TEXTLIST TL_LOG_LEVEL
  0 = 'TRACE'
  1 = 'DEBUG'
  2 = 'INFO'
  3 = 'WARN'
  4 = 'ERROR'
  5 = 'OFF'
   = ''
END_TEXTLIST

(* stored: Version 1.1.0.1, ProductVersion 3.1.4026.18
   TextList TL_LOG_LEVEL: Id {78f76045-66af-44f9-b46f-f8736d5f7626} *)
